// TIA Portal V20 export
TYPE "typeCmControlNodeSoftCam"
// stored: Namespace Unit1.Em5
   STRUCT
      manualInput { ExternalWritable := 'False'} : "Unit1.Em5.typeCmControlNodeSoftCamManualInput";
      magazine { ExternalWritable := 'False'} : "Unit1.Em5.typeCmControlNodeSoftCamMagazine";
   END_STRUCT;
END_TYPE
